(* IEC 61131-3 sources: repolevel_ST_code_completion/dataset/project_code/plc_hello_mixing_tank/FUN, 6 files *)

(* ---- F_ResetDeviceCommands.st ---- *)
FUNCTION F_ResetDeviceCommands : BOOL
VAR_IN_OUT
	// HMI命令标志（需要复位）
	bMixerRunCmd		:	BOOL;
	bMixerStopCmd		:	BOOL;
	bMedium1OpenCmd		:	BOOL;
	bMedium1CloseCmd	:	BOOL;
	bMedium2OpenCmd		:	BOOL;
	bMedium2CloseCmd	:	BOOL;
	bDrainOpenCmd		:	BOOL;
	bDrainCloseCmd		:	BOOL;
END_VAR
VAR_INPUT
	// 设备状态反馈
	bMixerRunning		:	BOOL;
	bMedium1Opened		:	BOOL;
	bMedium2Opened		:	BOOL;
	bDrainOpened		:	BOOL;
END_VAR

// 命令合理性复位
// 当设备到达目标状态时，复位相应的命令标志

// 混合电机命令复位
IF bMixerRunning THEN
	bMixerRunCmd := FALSE;		// 已运行，复位运行命令
ELSE
	bMixerStopCmd := FALSE;		// 已停止，复位停止命令
END_IF

// 介质1阀门命令复位
IF bMedium1Opened THEN
	bMedium1OpenCmd := FALSE;	// 已打开，复位打开命令
ELSE
	bMedium1CloseCmd := FALSE;	// 已关闭，复位关闭命令
END_IF

// 介质2阀门命令复位
IF bMedium2Opened THEN
	bMedium2OpenCmd := FALSE;	// 已打开，复位打开命令
ELSE
	bMedium2CloseCmd := FALSE;	// 已关闭，复位关闭命令
END_IF

// 排空阀门命令复位
IF bDrainOpened THEN
	bDrainOpenCmd := FALSE;		// 已打开，复位打开命令
ELSE
	bDrainCloseCmd := FALSE;	// 已关闭，复位关闭命令
END_IF

F_ResetDeviceCommands := TRUE;

(* ---- F_UpdateLimitSwitches.st ---- *)
FUNCTION F_UpdateLimitSwitches : BOOL
VAR_INPUT
	rTankLevel			:	REAL;			// 当前液位 (%)
	rFullThreshold		:	REAL := 85.0;	// 满液位阈值 (%)
	rEmptyThreshold		:	REAL := 5.0;	// 空液位阈值 (%)
END_VAR
VAR_OUTPUT
	bLevelFull			:	BOOL;			// 液位满开关
	bLevelEmpty			:	BOOL;			// 液位空开关
END_VAR

// 液位开关模拟
bLevelFull := rTankLevel >= rFullThreshold;		// 液位 >= 85% 时，满开关激活
bLevelEmpty := rTankLevel <= rEmptyThreshold;	// 液位 <= 5% 时，空开关激活

F_UpdateLimitSwitches := TRUE;

(* ---- FB_AutoSequence.st ---- *)
FUNCTION_BLOCK FB_AutoSequence
VAR_INPUT
	bEnable				:	BOOL;			// 使能自动序列
	bReset				:	BOOL;			// 复位到排空状态

	// 液位传感器反馈
	bTankLevelFull		:	BOOL;			// 液位满传感器
	bTankLevelEmpty		:	BOOL;			// 液位空传感器

	// 设备状态反馈
	bMixerRunning		:	BOOL;			// 混合电机运行中
	bMedium1Opened		:	BOOL;			// 介质1阀门打开
	bMedium2Opened		:	BOOL;			// 介质2阀门打开
	bDrainOpened		:	BOOL;			// 排空阀门打开

	// 配置参数
	tMixingDuration		:	TIME := T#10S;	// 混合持续时间
END_VAR
VAR_OUTPUT
	// 设备控制输出
	bMixerRunCmd		:	BOOL;			// 混合电机运行命令
	bMedium1OpenCmd		:	BOOL;			// 介质1阀门打开命令
	bMedium2OpenCmd		:	BOOL;			// 介质2阀门打开命令
	bDrainOpenCmd		:	BOOL;			// 排空阀门打开命令

	// 状态输出
	eCurrentState		:	AUTO_SEQUENCE;	// 当前状态
	nCyclesCompleted	:	UINT;			// 完成的循环次数
END_VAR
VAR
	tonMixing			:	TON;			// 混合定时器
END_VAR

// 复位逻辑
IF bReset THEN
	eCurrentState := AUTO_SEQUENCE.DRAINING;
	nCyclesCompleted := 0;
END_IF

// 自动序列状态机
IF bEnable THEN
	CASE eCurrentState OF
		AUTO_SEQUENCE.FILLING:
			// 确保其他设备不工作
			bMixerRunCmd := FALSE;
			bDrainOpenCmd := FALSE;

			// 打开两个介质阀门，开始填充罐体
			bMedium1OpenCmd := NOT bTankLevelFull;
			bMedium2OpenCmd := NOT bTankLevelFull;

			// 当罐体满时，等待填充阀关闭，然后进入混合状态
			IF bTankLevelFull AND NOT (bMedium1Opened OR bMedium2Opened) THEN
				eCurrentState := AUTO_SEQUENCE.MIXING;
			END_IF

		AUTO_SEQUENCE.MIXING:
			// 确保其他设备不工作
			bMedium1OpenCmd := FALSE;
			bMedium2OpenCmd := FALSE;
			bDrainOpenCmd := FALSE;

			// 启动混合电机并混合10秒
			bMixerRunCmd := TRUE;
			tonMixing(IN := bMixerRunning, PT := tMixingDuration);

			// 当定时器到达10秒，等待电机停止运行，然后进入排空状态
			IF tonMixing.Q THEN
				bMixerRunCmd := FALSE;
				eCurrentState := AUTO_SEQUENCE.DRAINING;
			END_IF

		AUTO_SEQUENCE.DRAINING:
			// 确保其他设备不工作
			bMixerRunCmd := FALSE;
			bMedium1OpenCmd := FALSE;
			bMedium2OpenCmd := FALSE;

			// 打开排空阀，开始排空罐体
			bDrainOpenCmd := NOT bTankLevelEmpty;

			// 当罐体空时，等待排空阀关闭，然后进入填充状态
			IF bTankLevelEmpty AND NOT bDrainOpened THEN
				eCurrentState := AUTO_SEQUENCE.FILLING;
				nCyclesCompleted := nCyclesCompleted + 1;
			END_IF
	END_CASE
ELSE
	// 禁用时，关闭所有输出
	bMixerRunCmd := FALSE;
	bMedium1OpenCmd := FALSE;
	bMedium2OpenCmd := FALSE;
	bDrainOpenCmd := FALSE;
	tonMixing(IN := FALSE);
END_IF

(* ---- FB_ManualControl.st ---- *)
FUNCTION_BLOCK FB_ManualControl
VAR_INPUT
	// HMI命令输入
	bMixerRunCmd		:	BOOL;
	bMixerStopCmd		:	BOOL;
	bMedium1OpenCmd		:	BOOL;
	bMedium1CloseCmd	:	BOOL;
	bMedium2OpenCmd		:	BOOL;
	bMedium2CloseCmd	:	BOOL;
	bDrainOpenCmd		:	BOOL;
	bDrainCloseCmd		:	BOOL;

	// 设备反馈输入
	bMixerRunning		:	BOOL;
	bMedium1Opened		:	BOOL;
	bMedium2Opened		:	BOOL;
	bDrainOpened		:	BOOL;
END_VAR
VAR_OUTPUT
	// 设备控制输出
	bMixerRunCmdOut		:	BOOL;
	bMedium1OpenCmdOut	:	BOOL;
	bMedium2OpenCmdOut	:	BOOL;
	bDrainOpenCmdOut	:	BOOL;
END_VAR

// 手动模式：HMI命令通过锁存器控制设备
// 锁存逻辑：按下启动OR已启动反馈 AND NOT 按下停止

// 混合电机控制
bMixerRunCmdOut := (bMixerRunCmd OR bMixerRunning) AND NOT bMixerStopCmd;

// 介质1阀门控制
bMedium1OpenCmdOut := (bMedium1OpenCmd OR bMedium1Opened) AND NOT bMedium1CloseCmd;

// 介质2阀门控制
bMedium2OpenCmdOut := (bMedium2OpenCmd OR bMedium2Opened) AND NOT bMedium2CloseCmd;

// 排空阀门控制
bDrainOpenCmdOut := (bDrainOpenCmd OR bDrainOpened) AND NOT bDrainCloseCmd;

(* ---- FB_ModeController.st ---- *)
FUNCTION_BLOCK FB_ModeController
VAR_INPUT
	bSetToAuto		:	BOOL;	// 切换到自动模式命令
	bSetToManual	:	BOOL;	// 切换到手动模式命令
END_VAR
VAR_OUTPUT
	eCurrentMode	:	MODES;	// 当前模式
	bModeChanged	:	BOOL;	// 模式改变标志
END_VAR
VAR
	eLastMode		:	MODES;	// 上次模式
END_VAR

// 模式切换逻辑
CASE eCurrentMode OF
	MODES.AUTO:
		IF bSetToManual THEN
			eCurrentMode := MODES.MANUAL;
		END_IF

	MODES.MANUAL:
		IF bSetToAuto THEN
			eCurrentMode := MODES.AUTO;
		END_IF
END_CASE

// 检测模式变化
bModeChanged := (eCurrentMode <> eLastMode);
eLastMode := eCurrentMode;

(* ---- FB_TankLevelSimulator.st ---- *)
FUNCTION_BLOCK FB_TankLevelSimulator
VAR_INPUT
	bMedium1Opened		:	BOOL;			// 介质1阀门打开
	bMedium2Opened		:	BOOL;			// 介质2阀门打开
	bDrainOpened		:	BOOL;			// 排空阀门打开
	bReset				:	BOOL;			// 复位到初始液位

	// 配置参数
	rInitialLevel		:	REAL := 25.0;	// 初始液位 (%)
	rFillRate1			:	REAL := 0.1;	// 介质1填充速率 (%/cycle)
	rFillRate2			:	REAL := 0.1;	// 介质2填充速率 (%/cycle)
	rDrainRate			:	REAL := 0.2;	// 排空速率 (%/cycle)
	rMinLevel			:	REAL := 0.0;	// 最小液位 (%)
	rMaxLevel			:	REAL := 100.0;	// 最大液位 (%)
END_VAR
VAR_OUTPUT
	rCurrentLevel		:	REAL;			// 当前液位 (%)
END_VAR

// 复位逻辑
IF bReset THEN
	rCurrentLevel := rInitialLevel;
END_IF

// 液位计算
// 如果任一填充阀打开则填充，如果排空阀打开则排空
rCurrentLevel := rCurrentLevel
				+ rFillRate1 * BOOL_TO_REAL(bMedium1Opened)
				+ rFillRate2 * BOOL_TO_REAL(bMedium2Opened)
				- rDrainRate * BOOL_TO_REAL(bDrainOpened);

// 限制液位范围 (0-100%)
rCurrentLevel := LIMIT(rMinLevel, rCurrentLevel, rMaxLevel);
